FUNCTION_BLOCK FB_PWM
VAR_INPUT
	pwmCycleTime 		: TIME := T#10S;
	pwmDutyCycle		: REAL := 0.5;
	reset				: BOOL := FALSE;
END_VAR
VAR_OUTPUT
	Q					: BOOL := FALSE;
END_VAR
VAR
	pwmTimeInMs			: INT	:= 0;
	pwmTimer		: TON;
	pwmLowTimer			: TON;
	dutyCycleInMs		: TIME;
	test				: INT;
	internalReset 		: BOOL := FALSE;
END_VAR

IF pwmDutyCycle < 0 THEN
	pwmDutyCycle := 0.0;
END_IF

IF reset OR internalReset THEN
	pwmTimer(IN:= FALSE);
	reset := FALSE;
	internalReset := FALSE;
ELSE
	pwmTimeInMs := TIME_TO_INT(pwmCycleTime);
	IF Q THEN
		(* high  --> running falling timer *)
		dutyCycleInMs := INT_TO_TIME(REAL_TO_INT(INT_TO_REAL(pwmTimeInMs)*pwmDutyCycle));
		pwmTimer(IN:=TRUE, PT:=dutyCycleInMs);
		IF pwmTimer.Q THEN
			internalReset := TRUE;
			Q := FALSE;
		END_IF		
	ELSE
		(* low --> running rising timer *)
		dutyCycleInMs := INT_TO_TIME(REAL_TO_INT(INT_TO_REAL(pwmTimeInMs)*(1.0-pwmDutyCycle)));
		pwmTimer(IN:=TRUE, PT:=dutyCycleInMs);
		IF pwmTimer.Q THEN
			internalReset := TRUE;
			Q := TRUE;
		END_IF		
	END_IF
END_IF

END_FUNCTION_BLOCK

(* stored: Version 1.1.0.1, ProductVersion 3.1.4022.7
   POU FB_PWM: Id {849a4c87-8406-4eb1-a849-917a58b91250}, SpecialFunc None *)
